(* CODESYS project SPT_Event_Logger.library
   Company: Beckhoff Automation LLC
   DefaultNamespace: SPT_EventLogger
   Version: 3.9.0
   Placeholder: SPT Event Logger
   Title: SPT Event Logger

Project tree, tasks and I/O mapping:
  libraries: Tc3_EventLogger, * (Beckhoff Automation GmbH); Tc3_Module, * (Beckhoff Automation GmbH)
  Project Information/
    function F_GetCompany [ST]
    function F_GetTitle [ST]
    function F_GetVersion [ST]
  Version/
    global variables Global_Version
  function F_ClearAllEventsInClass [ST]
  function F_CreateAllEventsInClass [ST]
  function F_GetMaxSeverityRaised [ST]
  function F_RaiseAlarm [ST]
  function F_RaiseAlarmAndSetFlags [ST]
  function F_RaiseAlarmWithStringParameters [ST]
  function F_RaiseAlarmWithStringsAndFlags [ST]
  00000000-0000-0000-0000-000000000000|LICENSE
  LICENSE
*)

// Version/Global_Version
{attribute 'TcGenerated'}
{attribute 'no-analysis'}
{attribute 'linkalways'}

// This function has been automatically generated from the project information.
VAR_GLOBAL CONSTANT
	{attribute 'const_non_replaced'}
	stLibVersion_SPT_Event_Logger : ST_LibVersion := (iMajor := 3, iMinor := 9, iBuild := 0, iRevision := 0, nFlags := 0, sVersion := '3.9.0');
END_VAR

// Project Information/F_GetCompany
// This function has been automatically generated from the project information.
{attribute 'signature_flag' := '1073741824'}
{attribute 'TcGenerated'}
{attribute 'no-analysis'}
FUNCTION F_GetCompany : WSTRING
VAR_INPUT
	
END_VAR

F_GetCompany := "Beckhoff Automation LLC";

END_FUNCTION

// Project Information/F_GetTitle
// This function has been automatically generated from the project information.
{attribute 'signature_flag' := '1073741824'}
{attribute 'TcGenerated'}
{attribute 'no-analysis'}
FUNCTION F_GetTitle : WSTRING
VAR_INPUT
	
END_VAR

F_GetTitle := "SPT Event Logger";

END_FUNCTION

// Project Information/F_GetVersion
// This function has been automatically generated from the project information.
{attribute 'signature_flag' := '1073741824'}
{attribute 'TcGenerated'}
{attribute 'no-analysis'}
FUNCTION F_GetVersion : ST_LibVersion
VAR_INPUT
	
END_VAR

F_GetVersion.iMajor := 3;
F_GetVersion.iMinor := 9;
F_GetVersion.iBuild := 0;
F_GetVersion.iRevision := 0;
F_GetVersion.sVersion := '3.9.0';
F_GetVersion.nFlags := 1;

END_FUNCTION

// F_ClearAllEventsInClass
// Initializes event function blocks for an entire event class using auto-generated source info
FUNCTION F_ClearAllEventsInClass
VAR_IN_OUT
	Alarms : ARRAY[*] OF FB_TcAlarm; // Array of Alarms to be defined
END_VAR

VAR
	i : DINT;
END_VAR

FOR i := LOWER_BOUND(Alarms, 1) TO UPPER_BOUND(Alarms, 1) DO
	IF Alarms[i].bRaised THEN
		Alarms[i].Clear(0, 0);
	END_IF
END_FOR

END_FUNCTION

// F_CreateAllEventsInClass
// Initializes event function blocks for an entire event class using auto-generated source info
FUNCTION F_CreateAllEventsInClass
VAR_IN_OUT
	Alarms : ARRAY[*] OF FB_TcAlarm; // Array of Alarms to be defined
END_VAR

VAR_INPUT
	ClassSize  : UDINT;					  // Size in bytes of the event class
	pInitEvent : POINTER TO TcEventEntry; // Address of first event in Event Class (Should be the InitReferenceEvent)
	Prefix	   : STRING;				  // String Prefix for the Event Message -- Usually the Module ID and Name
END_VAR

VAR
	i			   : UDINT;
	EventSize	   : UDINT;
	numberOfEvents : UDINT;
	pEvent		   : POINTER TO TcEventEntry;
END_VAR

EventSize	   := SIZEOF(pInitEvent^);
numberOfEvents := ClassSize / EventSize;
FOR i := TO_UDINT(LOWER_BOUND(Alarms, 1)) TO TO_UDINT(UPPER_BOUND(Alarms, 1)) DO
	IF i > numberOfEvents THEN
		EXIT;
	ELSE
		pEvent := pInitEvent + ((i - 1) * EventSize);
		Alarms[i].CreateEx(stEventEntry := pEvent^, 0, 0);
		Alarms[i].ipArguments.AddString(Prefix);
	END_IF
END_FOR

END_FUNCTION

// F_GetMaxSeverityRaised
// Compares a collection of alarms to current alarm severity and returns the maximum severity of any raised alarm
FUNCTION F_GetMaxSeverityRaised : TcEventSeverity // Maximum severity
VAR_IN_OUT
	Alarms : ARRAY[*] OF FB_TcAlarm; // Events to compare against
END_VAR

VAR_INPUT
	CurrentSeverity : TcEventSeverity; // Current severity of module alarm
END_VAR

VAR
	i : DINT;
END_VAR

FOR i := LOWER_BOUND(Alarms, 1) TO UPPER_BOUND(Alarms, 1) DO
	IF Alarms[i].bRaised AND (Alarms[i].eSeverity > CurrentSeverity) THEN
		CurrentSeverity := Alarms[i].eSeverity;
	END_IF
END_FOR

F_GetMaxSeverityRaised := CurrentSeverity;

END_FUNCTION

// F_RaiseAlarm
// Raises an alarm and sets fault info to variables which are passed in
FUNCTION F_RaiseAlarm
VAR_IN_OUT
	Alarm : FB_TcAlarm; // Alarm to be raised
END_VAR

IF NOT Alarm.bRaised THEN
	Alarm.Raise(0);
END_IF

END_FUNCTION

// F_RaiseAlarmAndSetFlags
// Raises an alarm and sets fault info to variables which are passed in
FUNCTION F_RaiseAlarmAndSetFlags
VAR_IN_OUT
	Alarm	  : FB_TcAlarm; // Alarm to be raised
	ErrorFlag : BOOL;		// Error flag to set (VAR_IN_OUT, put the variable you want the function to SET here)
	ErrorID	  : UDINT;		// Error ID to set (VAR_IN_OUT, put the variable you want the function to SET here) - Will be set using the ID of the given fbAlarm
END_VAR

ErrorFlag := TRUE;
ErrorID	  := Alarm.nEventId;
Alarm.Raise(0);

END_FUNCTION

// F_RaiseAlarmWithStringParameters
// Raises an alarm and passes string arguments as parameters for extra fault context/info
FUNCTION F_RaiseAlarmWithStringParameters
VAR_IN_OUT
	Alarm : FB_TcAlarm; // Alarm to be raised
END_VAR

VAR_INPUT
	String_1 : STRING; // First string parameter
	String_2 : STRING; // Second string parameter
	String_3 : STRING; // Third string parameter
END_VAR

Alarm.ipArguments.Clear();
IF String_1 <> '' THEN
	Alarm.ipArguments.AddString(String_1);
END_IF

IF String_2 <> '' THEN
	Alarm.ipArguments.AddString(String_2);
END_IF

IF String_3 <> '' THEN
	Alarm.ipArguments.AddString(String_3);
END_IF

Alarm.Raise(0);

END_FUNCTION

// F_RaiseAlarmWithStringsAndFlags
// Raises an alarm and passes string arguments as parameters for extra fault context/info. Additionally sets fault info to variables which are passed in
FUNCTION F_RaiseAlarmWithStringsAndFlags
VAR_IN_OUT
	Alarm	  : FB_TcAlarm; // Alarm to be raised
	ErrorFlag : BOOL;		// Error flag to set (VAR_IN_OUT, put the variable you want the function to SET here)
	ErrorID	  : UDINT;		// Error ID to set (VAR_IN_OUT, put the variable you want the function to SET here) - Will be set using the ID of the given fbAlarm
END_VAR

VAR_INPUT
	String_1 : STRING; // First string parameter
	String_2 : STRING; // Second string parameter
	String_3 : STRING; // Third string parameter
END_VAR

Alarm.ipArguments.Clear();
ErrorFlag := TRUE;
ErrorID	  := Alarm.nEventId;
F_RaiseAlarmWithStringParameters(Alarm	  := Alarm,
								 String_1 := String_1,
								 String_2 := String_2,
								 String_3 := String_3);

END_FUNCTION
